(* PLC project ARR NG V1.0, SoMachine Motion Logic Builder V1.56.49.0, author SESA100920 *)
(* stored: creationDateTime 2020-05-25T16:32:27.539003, version 0.0.0.0, modificationDateTime 2020-05-15T14:58:38.6738722 *)

PROGRAM DigitalTwin
  VAR
    sIp : STRING(15) := '10.139.10.6';
    uiPort : UINT := 5005;
    fbUdpPeer : TCPUDP.FB_UDPPeer;
    uiVal1 : UINT;
    uiVal2 : UINT;
    uiVal3 : UINT;
    uiVal4 : UINT;
    uiVal5 : UINT;
    uiVal6 : UINT;
    uiVal7 : UINT;
    uiVal8 : UINT;
    s1 : STRING;
    s2 : STRING;
    s3 : STRING;
    s4 : STRING;
    s5 : STRING;
    s6 : STRING;
    s7 : STRING;
    s8 : STRING;
    sStringToSend : STRING;
    udiSize : UDINT;
    iVal : INT;
  END_VAR

            CASE iVal OF
	0: IF fbUdpPeer.Open() THEN
		iVal := 1;
		END_IF
	1: 
		uiVal1 := LREAL_TO_UINT(DRV_Robot1_A.Position);
		uiVal2 := LREAL_TO_UINT(DRV_Robot1_B.Position);
		uiVal3 := LREAL_TO_UINT(DRV_Robot1_C.Position);
		uiVal4 := LREAL_TO_UINT(DRV_Robot2_A.Position);
		uiVal5 := LREAL_TO_UINT(DRV_Robot2_B.Position);
		uiVal6 := LREAL_TO_UINT(DRV_Robot2_C.Position);
		uiVal7 := LREAL_TO_INT(DRV_Robot1_AuxAx1.Position);
		uiVal8 := LREAL_TO_INT(DRV_Robot2_AuxAx1.Position);
		s1 := UINT_TO_STRING(uiVal1);
		s2 := UINT_TO_STRING(uiVal2);
		s3 := UINT_TO_STRING(uiVal3);
		s4 := UINT_TO_STRING(uiVal4);
		s5 := UINT_TO_STRING(uiVal5);
		s6 := UINT_TO_STRING(uiVal6);
		s7 := UINT_TO_STRING(uiVal7);
		s8 := UINT_TO_STRING(uiVal8);
		s1 := CONCAT('X',s1);
		s2 := CONCAT('Y',s2);
		s3 := CONCAT('Z',s3);
		s4 := CONCAT('X',s4);
		s5 := CONCAT('Y',s5);
		s6 := CONCAT('Z',s6);
		s7 := CONCAT('A',s7);
		s8 := CONCAT('B',s8);
		sStringToSend := CONCAT(CONCAT(CONCAT(s1,s2), CONCAT(s3,s4)), CONCAT(CONCAT(s5,s6), CONCAT(s7,s8)));
		udiSize := SIZEOF(sStringToSend);
		fbUdpPeer.SendTo(sIp, uiPort, ADR(sStringToSend), udiSize);		
END_CASE
          
END_PROGRAM
